// TIA Portal project "AutoII-G1" (V16)

(* hardware
DEVICE "S7-1200 station_1"  S7-1200 Station
   slot 0: "Rack_0"  S7-1200 Rack  Rack  V1.0
   slot 1: "PLC_1"  CPU 1214C DC/DC/DC  6ES7 214-1AG40-0XB0  V4.4
   slot 2: "DI 16/DQ 16x24VDC_1"  6ES7 223-1BL32-0XB0  V2.0
*)

// ===== PLC "PLC_1"  CPU 1214C DC/DC/DC =====

VAR_GLOBAL   // PLC tag table "Tabla de variables estándar"
   "ARRANQUE_M1" AT %I0.0 : Bool;
   "PARO_M1" AT %I0.1 : Bool;
   "FALLA_M1" AT %I0.2 : Bool;
   "MOTOR1" AT %Q0.0 : Bool;
   "ARRANQUE_M2" AT %I0.3 : Bool;
   "PARO_M2" AT %I0.4 : Bool;
   "FALLA_M2" AT %I0.5 : Bool;
   "MOTOR2" AT %Q0.1 : Bool;
   "ARRANQUE_M3" AT %I0.6 : Bool;
   "PARO_M3" AT %I0.7 : Bool;
   "FALLA_M3" AT %I1.0 : Bool;
   "MOTOR3" AT %Q0.2 : Bool;
   "Tag_1" AT %M0.0 : Bool;
   "Tag_2" AT %M0.1 : Bool;
   "Tag_3" AT %M0.2 : Bool;
   "Abrir_V1" AT %I2.0 : Bool;
   "Cerrar_V1" AT %I2.1 : Bool;
   "Q_Abrir_V1" AT %Q2.0 : Bool;
   "Aux_V1" AT %M2.0 : Bool;
   "Tag_4" AT %Q0.3 : Bool;
   "Conf_Ab_V1" AT %I2.2 : Bool;
   "Conf_Cer_V1" AT %I2.3 : Bool;
   "Q_Cerrar_V1" AT %Q2.1 : Bool;
END_VAR

DATA_BLOCK "VALVULA_V1"   // DB3
{ S7_Optimized_Access := 'TRUE' }
VERSION : 0.1
// stored: InstanceOfName VALVULA
"VALVULA"
BEGIN
END_DATA_BLOCK

// folder: System blocks/Program resources

DATA_BLOCK "T_ON_M2"   // DB1
{ S7_Optimized_Access := 'TRUE' }
AUTHOR : Simatic
FAMILY : IEC
NAME : IEC_TMR
VERSION : 1.0
// stored: InstanceOfName IEC_TIMER
"IEC_TIMER"
BEGIN
END_DATA_BLOCK

DATA_BLOCK "T_ON_M3"   // DB2
{ S7_Optimized_Access := 'TRUE' }
AUTHOR : Simatic
FAMILY : IEC
NAME : IEC_TMR
VERSION : 1.0
// stored: InstanceOfName IEC_TIMER
"IEC_TIMER"
BEGIN
END_DATA_BLOCK

// folder: (top level)

FUNCTION_BLOCK "VALVULA"   // FB1, LAD
{ S7_Optimized_Access := 'TRUE' }
VERSION : 0.1
   VAR_INPUT
      Abrir : Bool;
      Conf_Abierta : Bool;
      Hab_Conf_Ab : Bool;
      T_Abrir : Time;
      Cerrar : Bool;
      Conf_Cerrada : Bool;
      Hab_Conf_Cer : Bool;
      T_Cierre : Time;
   END_VAR
   VAR_OUTPUT
      Q_Abrir : Bool;
      Q_Cerrar : Bool;
   END_VAR
   VAR
      Aux_Valvula : Bool;
      Aux_Valvula2 : Bool;
      TP_Cierre : IEC_TIMER;
      TP_Abrir : IEC_TIMER;
   END_VAR
BEGIN

REGION Network 1
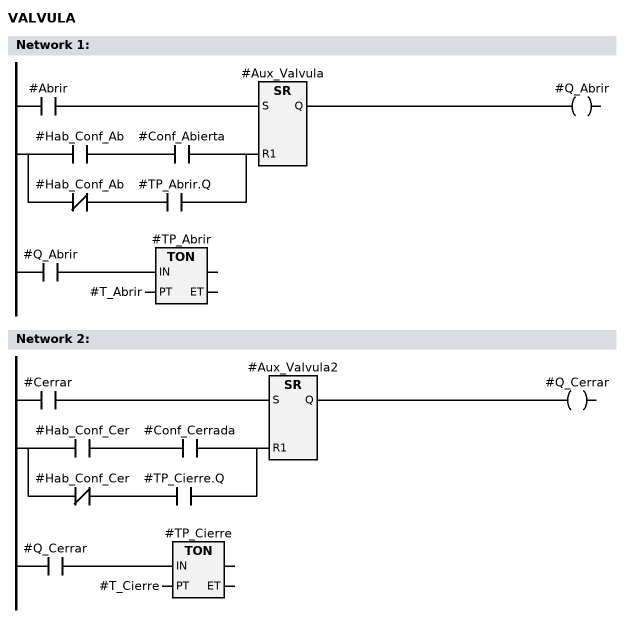
   IF #Abrir THEN
       #Aux_Valvula := TRUE;   // SR flip-flop
   END_IF;
   IF (#Hab_Conf_Ab AND #Conf_Abierta) OR (NOT #Hab_Conf_Ab AND #TP_Abrir.Q) THEN
       #Aux_Valvula := FALSE;
   END_IF;
   #Q_Abrir := #Aux_Valvula;
   #TP_Abrir.TON(IN := #Q_Abrir, PT := #T_Abrir);
END_REGION

REGION Network 2
   IF #Cerrar THEN
       #Aux_Valvula2 := TRUE;   // SR flip-flop
   END_IF;
   IF (#Hab_Conf_Cer AND #Conf_Cerrada) OR (NOT #Hab_Conf_Cer AND #TP_Cierre.Q) THEN
       #Aux_Valvula2 := FALSE;
   END_IF;
   #Q_Cerrar := #Aux_Valvula2;
   #TP_Cierre.TON(IN := #Q_Cerrar, PT := #T_Cierre);
END_REGION
END_FUNCTION_BLOCK

FUNCTION "MOTOR" : Void   // FC1, LAD
{ S7_Optimized_Access := 'TRUE' }
VERSION : 0.1
   VAR_INPUT
      ARRANQUE : Bool;
      PARO : Bool;
      FALLA : Bool;
   END_VAR
   VAR_OUTPUT
      MOTOR : Bool;
   END_VAR
   VAR_IN_OUT
      mARRANQUE : Bool;
   END_VAR
BEGIN

REGION Network 1
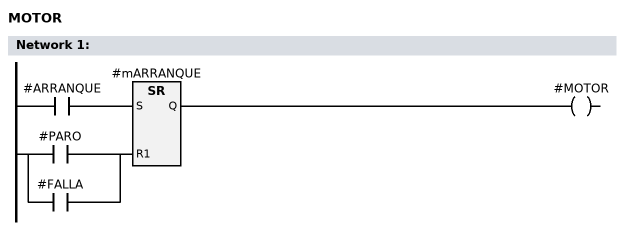
   RUNG wire#powerrail
      Contact( #ARRANQUE )
      S_SR(operand := #mARRANQUE, r1 := wire#w1)
      Coil( #MOTOR )
   END_RUNG
   RUNG wire#powerrail
      Contact( #PARO )
   END_RUNG wire#w1
   RUNG wire#powerrail
      Contact( #FALLA )
   END_RUNG wire#w1
   // the same network as SCL:
   IF #ARRANQUE THEN
       #mARRANQUE := TRUE;   // SR flip-flop
   END_IF;
   IF #PARO OR #FALLA THEN #mARRANQUE := FALSE; END_IF;
   #MOTOR := #mARRANQUE;
END_REGION
END_FUNCTION

ORGANIZATION_BLOCK "Main"   // OB1, LAD, ProgramCycle
TITLE = "Main Program Sweep (Cycle)"
{ S7_Optimized_Access := 'TRUE' }
VERSION : 0.1
BEGIN

REGION Network 1
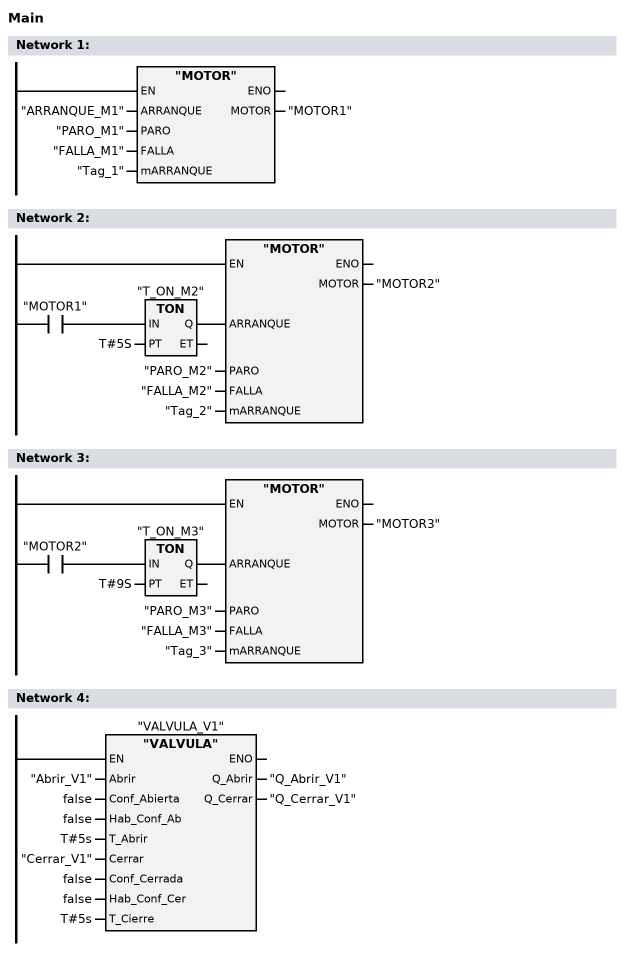
   RUNG wire#powerrail
      "MOTOR"(ARRANQUE := "ARRANQUE_M1", PARO := "PARO_M1", FALLA := "FALLA_M1", mARRANQUE := "Tag_1", MOTOR => "MOTOR1")
   END_RUNG
   // the same network as SCL:
   "MOTOR"(ARRANQUE := "ARRANQUE_M1",
           PARO := "PARO_M1",
           FALLA := "FALLA_M1",
           mARRANQUE := "Tag_1",
           MOTOR => "MOTOR1");
END_REGION

REGION Network 2
   "T_ON_M2".TON(IN := "MOTOR1", PT := T#5S);
   "MOTOR"(ARRANQUE := "T_ON_M2".Q,
           PARO := "PARO_M2",
           FALLA := "FALLA_M2",
           mARRANQUE := "Tag_2",
           MOTOR => "MOTOR2");
END_REGION

REGION Network 3
   "T_ON_M3".TON(IN := "MOTOR2", PT := T#9S);
   "MOTOR"(ARRANQUE := "T_ON_M3".Q,
           PARO := "PARO_M3",
           FALLA := "FALLA_M3",
           mARRANQUE := "Tag_3",
           MOTOR => "MOTOR3");
END_REGION

REGION Network 4
   RUNG wire#powerrail
      "VALVULA_V1"(Abrir := "Abrir_V1", Conf_Abierta := false, Hab_Conf_Ab := false, T_Abrir := T#5s, Cerrar := "Cerrar_V1", Conf_Cerrada := false, Hab_Conf_Cer := false, T_Cierre := T#5s, Q_Abrir => "Q_Abrir_V1", Q_Cerrar => "Q_Cerrar_V1")
   END_RUNG
   // the same network as SCL:
   "VALVULA_V1"(Abrir := "Abrir_V1",   // "VALVULA"
                Conf_Abierta := false,
                Hab_Conf_Ab := false,
                T_Abrir := T#5s,
                Cerrar := "Cerrar_V1",
                Conf_Cerrada := false,
                Hab_Conf_Cer := false,
                T_Cierre := T#5s,
                Q_Abrir => "Q_Abrir_V1",
                Q_Cerrar => "Q_Cerrar_V1");
END_REGION
END_ORGANIZATION_BLOCK